(*
version 1.1	16 sep 2007
programmer 	hugo
tested by		tobias

FT_TN16 is delay function, it will delay a signal by a specified time : T and will store 16 values of in before they are put thru to out.
for higher or lower resolution please use FT_TN8 or FT_TN64 instead.

*)
FUNCTION_BLOCK FT_TN16
VAR_INPUT
	in : REAL;
	T : TIME;
END_VAR
VAR_OUTPUT
	out : REAL;
	trig : BOOL;
END_VAR
VAR
	length : INT := 16;
	X : ARRAY[0..15] OF REAL;
	cnt : INT;
	last : TIME;
	tx: TIME;
	init: BOOL;
END_VAR

(* read system time *)
tx := DWORD_TO_TIME(T_PLC_MS());

trig := FALSE;
IF NOT init THEN
	x[cnt] := in;
	init := TRUE;
	last := tx;
ELSIF tx - last >= T / length THEN
	IF cnt = length - 1 THEN cnt := 0; ELSE cnt := cnt + 1; END_IF;
	Out := X[cnt];
	x[cnt] := in;
	last := tx;
	Trig := TRUE;
END_IF;

(* revision history
hm		1. jan 2007	rev 1.0
	original version

hm		16. sep 2007	rev 1.1
	changes time() to T_plc_ms() for compatibility reasons

*)

END_FUNCTION_BLOCK

(* stored: Version 1.1.0.1
   POU FT_TN16: Id {52d08263-28ee-49b7-b06d-9004585144d2}, SpecialFunc None *)
